INTERFACE IDrive

METHOD MoveAbsolute : TcoCore.ITcoTaskStatus
VAR_INPUT
	TargetPosition : LREAL;
END_VAR
END_METHOD

PROPERTY MoveAbsoluteTask : REFERENCE TO DriveSimMoveAbsoluteTask
GET
END_GET
END_PROPERTY

END_INTERFACE

(* stored: Version 1.1.0.1, ProductVersion 3.1.4024.9
   Itf IDrive: Id {56a4a9b0-da64-4b93-9928-f728021459b0}
   Method MoveAbsolute: Id {c317d00a-5ad5-412f-88c4-709bf3587e00}
   Property MoveAbsoluteTask: Id {c8fdae37-d359-4d29-8433-5d3fa1a2d1a9}
   Get Get: Id {1282b1a0-8dd1-4c95-b04e-7c5bcb844aca} *)
